TYPE E_Mode :
(
	OFF := 1,
	Manual,
	Auto
)USINT;
END_TYPE

(* stored: Version 1.1.0.1, ProductVersion 3.1.4024.12
   DUT E_Mode: Id {5e68e5a8-56a0-470f-93d0-1912672b3b3f} *)
